TYPE SetPointAdjustment :
STRUCT
	X: LREAL;
	Y: LREAL;
	Curve: SetPointOffsetCurve;
END_STRUCT
END_TYPE

(* stored: Version 1.1.0.1, ProductVersion 3.1.4024.6
   DUT SetPointAdjustment: Id {66e8ab10-f6e2-4cd9-b9cd-17f787b5ca44} *)
